{attribute 'linkalways'} 
{attribute 'no_explicit_call' := 'This FB is a CLASS and must be accessed using methods or properties'}
{attribute 'enable_dynamic_creation'}
FUNCTION_BLOCK Node_F_VN_AppendToContainer_TcVnRotatedRectangle EXTENDS VisionNode
VAR
    stElement : _TcVnRotatedRectangle;
    ipContainer : _ITcVnContainer;
    hrPrev : _HRESULT(S_OK);
	hresult : _HRESULT(S_OK);
END_VAR

METHOD PUBLIC  Clone : I_Node
VAR
	pNode : POINTER TO Node_F_VN_AppendToContainer_TcVnRotatedRectangle;
END_VAR
pNode := __NEW(Node_F_VN_AppendToContainer_TcVnRotatedRectangle);
Clone := pNode^;
END_METHOD

METHOD FB_init : BOOL
VAR_INPUT
	bInitRetains : BOOL; // if TRUE, the retain variables are initialized (warm start / cold start)
	bInCopyCode : BOOL;  // if TRUE, the instance afterwards gets moved into the copy code (online change)
END_VAR
AddInput('stElement', stElement);
AddInput('ipContainer', ipContainer);
AddInput('hrPrev', hrPrev);
AddOutput('ipContainer', ipContainer);
AddOutput('hresult',hresult);
END_METHOD

METHOD PROTECTED OnExecute
hresult.Value := F_VN_AppendToContainer_TcVnRotatedRectangle(
    stElement := stElement.Value,
	ipContainer := ipContainer.Value,
	hrPrev:= hrPrev.Value);
END_METHOD

METHOD PUBLIC PreExecutionCheck
VAR_INPUT
	Check : I_PreExecutionChecks;
END_VAR
Check.IsTrue(ipContainer.IsValid, 'ipContainer must be a valid container');
Check.IsTrue(ipContainer.HasType(TC_GLOBAL_CONST_LIST.ContainerType_Vector_TcVnRotatedRectangle), 'ipContainer contains incorrect type');
END_METHOD

END_FUNCTION_BLOCK

(* stored: Version 1.1.0.1, ProductVersion 3.1.4024.15
   POU Node_F_VN_AppendToContainer_TcVnRotatedRectangle: Id {d0387417-aeb4-0cf5-12b1-fdde5689eae4}, SpecialFunc None
   Folder Constructor: Id {e83d0df6-c933-03d6-101b-4a559ff43b42}
   Method Clone: Id {246bada4-ad9e-083c-1657-adc71c8ee7d0}
   Method FB_init: Id {fca25367-08a0-0362-28c6-7a9b20cdd515}
   Method OnExecute: Id {9a2c0671-5a7d-01af-09df-7bb841699a25}
   Method PreExecutionCheck: Id {7f2c5f52-83b8-05ce-382d-ded44108ee7b} *)
